FUNCTION_BLOCK FB_Logger IMPLEMENTS I_Logger
VAR_INPUT
END_VAR
VAR_OUTPUT
END_VAR
VAR
END_VAR

METHOD PUBLIC M_Log
END_METHOD

END_FUNCTION_BLOCK

(* stored: Version 1.1.0.1
   POU FB_Logger: Id {55e334a1-890f-4fb0-98ef-c532b69ee1fd}, SpecialFunc None
   Method M_Log: Id {a9f6c2b8-bade-4429-b19a-5b07e920fc4a} *)
